(* IEC 61131-3 sources: volt/packages/volt-lsp-iec/test-corpus/CodesysTestProject/Device/Plc Logic/Application/Library Manager/(unresolved)/iodriver profibus2 interfaces, 16 files *)

(* ---- DP_STATIONSTATUS1.dut ---- *)
TYPE DP_STATIONSTATUS1 :
UNION
	VALUE : BYTE;
	DIAG : DP_StationStatus1_Diag;
END_UNION
END_TYPE

(* ---- DP_STATIONSTATUS1_DIAG.dut ---- *)
TYPE DP_STATIONSTATUS1_DIAG :
STRUCT
	STATION_NON_EXISTENT : BIT;
	STATION_NOT_READY : BIT;
	CFG_FAULT : BIT;
	EXT_DIAG : BIT;
	NOT_SUPPORTED : BIT;
	INVALID_SLAVE_RESPONSE : BIT;
	PRM_FAULT : BIT;
	MASTER_LOCK : BIT;
END_STRUCT
END_TYPE

(* ---- DP_STATIONSTATUS2.dut ---- *)
TYPE DP_STATIONSTATUS2 :
UNION
	VALUE : BYTE;
	DIAG : DP_StationStatus2_Diag;
END_UNION
END_TYPE

(* ---- DP_STATIONSTATUS2_DIAG.dut ---- *)
TYPE DP_STATIONSTATUS2_DIAG :
STRUCT
	PRM_REQ : BIT;
	STAT_DIAG : BIT;
	DP : BIT;
	WD_ON : BIT;
	FREEZE_MODE : BIT;
	SYNC_MODE : BIT;
	RESERVED : BIT;
	DEACTIVATED : BIT;
END_STRUCT
END_TYPE

(* ---- DP_STATIONSTATUS3.dut ---- *)
TYPE DP_STATIONSTATUS3 :
UNION
	VALUE : BYTE;
	DIAG : DP_StationStatus3_Diag;
END_UNION
END_TYPE

(* ---- DP_STATIONSTATUS3_DIAG.dut ---- *)
TYPE DP_STATIONSTATUS3_DIAG :
STRUCT
	RESERVED0 : BIT;
	RESERVED1 : BIT;
	RESERVED2 : BIT;
	RESERVED3 : BIT;
	RESERVED4 : BIT;
	RESERVED5 : BIT;
	RESERVED6 : BIT;
	EXT_DIAG_OVERFLOW : BIT;
END_STRUCT
END_TYPE

(* ---- DPSLAVEDIAG.dut ---- *)
TYPE DPSLAVEDIAG :
STRUCT
	STATUS1 : DP_StationStatus1;
	STATUS2 : DP_StationStatus2;
	STATUS3 : DP_StationStatus3;
	DIAG_MASTER_ADD : USINT;
	IDENT_NUMBER : UINT;
END_STRUCT
END_TYPE

(* ---- PB_SLAVEACTIVATION.dut ---- *)
TYPE PB_SLAVEACTIVATION :
STRUCT
	XENABLE : BOOL;
	BYSTATIONADDRESS : BYTE;
	UDISLAVEACTIVAION : UDINT;
	WOPSTATE : WORD;
	UDIERROR : UDINT;
	UDIJOBID : UDINT;
	XENABLEOLD : BOOL;
	PCONNECTOR : POINTER TO BYTE;
	NCOUNT : DINT;
END_STRUCT
END_TYPE

(* ---- PB_SLAVECONFIGURATIONDATA.dut ---- *)
TYPE PB_SLAVECONFIGURATIONDATA :
STRUCT
	XENABLE : BOOL;
	BYSTATIONADDRESS : BYTE;
	PBYDATAAREA : POINTER TO BYTE;
	UDIDATASIZE : UDINT;
	WOPSTATE : WORD;
	UDICONFIGSIZE : UDINT;
	UDIERROR : UDINT;
	UDIJOBID : UDINT;
	XENABLEOLD : BOOL;
END_STRUCT
END_TYPE

(* ---- INTERFACEIDS.gvl ---- *)
VAR_GLOBAL
	ITFID_ICMPIODRVPROFIBUS : DWORD := 16#32;
	ITFID_ICMPIODRVPBSLAVEACTIVATION : DWORD := 16#50;
	ITFID_ICMPIODRVPROFIBUSCONFIG : DWORD := 16#5A;
END_VAR

(* ---- OPERATIONSTATES.gvl ---- *)
VAR_GLOBAL
	PB_NOT_ENABLED : WORD := 0;
	PB_INVALID_PARAMETER : WORD := 1;
	PB_PENDING : WORD := 2;
	PB_DONE : WORD := 3;
	PB_ERROR : WORD := 4;
END_VAR

(* ---- SLAVEACTIVATIONCOMMANDS.gvl ---- *)
VAR_GLOBAL
	PB_SLAVE_ACTIVE : UDINT := 0;
	PB_SLAVE_INACTIVE : UDINT := 1;
END_VAR

(* ---- ICMPIODRVPBSLAVEACTIVATION.itf ---- *)
INTERFACE ICMPIODRVPBSLAVEACTIVATION
END_INTERFACE

METHOD GETSLAVEACTIVATION : UDINT
VAR_IN_OUT
	TSLAVEACTIVATION : PB_SlaveActivation;
END_VAR
END_METHOD

METHOD SETSLAVEACTIVATION : UDINT
VAR_IN_OUT
	TSLAVEACTIVATION : PB_SlaveActivation;
END_VAR
END_METHOD

(* ---- ICMPIODRVPROFIBUS.itf ---- *)
INTERFACE ICMPIODRVPROFIBUS
END_INTERFACE

METHOD CLEARDATA : UDINT
VAR_INPUT
	UDIREMADR : UDINT;
	UDIGROUPSELECT : UDINT;
END_VAR
END_METHOD

METHOD FREEZE : UDINT
VAR_INPUT
	UDIREMADR : UDINT;
	UDIGROUPSELECT : UDINT;
END_VAR
END_METHOD

METHOD SYNC : UDINT
VAR_INPUT
	UDIREMADR : UDINT;
	UDIGROUPSELECT : UDINT;
END_VAR
END_METHOD

METHOD UNSYNC : UDINT
VAR_INPUT
	UDIREMADR : UDINT;
	UDIGROUPSELECT : UDINT;
END_VAR
END_METHOD

METHOD UNFREEZE : UDINT
VAR_INPUT
	UDIREMADR : UDINT;
	UDIGROUPSELECT : UDINT;
END_VAR
END_METHOD

(* ---- ICMPIODRVPROFIBUSCONFIG.itf ---- *)
INTERFACE ICMPIODRVPROFIBUSCONFIG
END_INTERFACE

METHOD GETSLAVECONFIGURATION : UDINT
VAR_IN_OUT
	TGETSLAVECONFIG : PB_SlaveConfigurationData;
END_VAR
END_METHOD

(* ---- IPBSLAVEDIAG.itf ---- *)
INTERFACE IPBSLAVEDIAG
END_INTERFACE

METHOD GETDIAG : DPSlaveDiag
END_METHOD

METHOD GETEXTDIAG : UINT
VAR_INPUT
	PEXTDIAG : POINTER TO BYTE;
	UIMAXLEN : UINT;
END_VAR
END_METHOD
